INTERFACE I_ListAssert

METHOD M_Add : BOOL
VAR_INPUT
	eAssert:		E_Assert;
	sMessage:		STRING(255);
	sType:			STRING(255);
END_VAR
END_METHOD

METHOD M_Clear
END_METHOD

METHOD M_Get : ST_Assert
VAR_INPUT
	nIndex: 	DINT;
END_VAR
END_METHOD

METHOD M_Index : DINT
VAR_INPUT
	eAssert:		E_Assert;
	sMessage:		STRING(255);
	sType:			STRING(255);
END_VAR
END_METHOD

METHOD M_Remove : BOOL
VAR_INPUT
	eAssert:		E_Assert;
	sMessage:		STRING(255);
	sType:			STRING(255);
END_VAR
END_METHOD

METHOD M_Search : DINT
VAR_INPUT
	eAssert:		E_Assert;
	sMessage:		STRING(255);
	sType:			STRING(255);
END_VAR
END_METHOD

PROPERTY P_Length : DINT
GET
END_GET
END_PROPERTY

END_INTERFACE

(* stored: Version 1.1.0.1
   Itf I_ListAssert: Id {937c5750-ac4a-0c75-3ddd-b288d095682e}
   Method M_Add: Id {3e064770-ed70-0084-0d0c-06375eeb81ec}
   Method M_Clear: Id {45d374a7-42f8-0c31-0d94-2816ec7b6d3b}
   Method M_Get: Id {a1dcf951-8b9f-0ae7-3dea-0f30a026ed8e}
   Method M_Index: Id {6b7196d0-67ec-0128-2e70-383439634955}
   Method M_Remove: Id {093efa55-1aa5-0156-0a6b-89b8a5b4082d}
   Method M_Search: Id {5c4d0ea8-2862-0b5d-1c53-fda70a30859a}
   Property P_Length: Id {dd1a731e-7c76-0405-3a5b-64fd53e98745}
   Get Get: Id {59abc2b2-589e-0023-0109-6a75ba5d563a} *)
